# EPICS autosave request: FOFBApp/Db/FOFBRtm_settings.req
$(P)$(R)RtmLampDacDataFromWb-SP
$(P)$(R)RtmLampAmpEn$(RTM_CHAN)-SP
$(P)$(R)RtmLampPIOLTriangEn$(RTM_CHAN)-SP
$(P)$(R)RtmLampPIOLSquareEn$(RTM_CHAN)-SP
$(P)$(R)RtmLampPISPSquareEn$(RTM_CHAN)-SP
$(P)$(R)RtmLampPIEn$(RTM_CHAN)-SP
$(P)$(R)RtmLampDacData$(RTM_CHAN)-SP
$(P)$(R)RtmLampDacWr$(RTM_CHAN)-SP
$(P)$(R)RtmLampPIKP$(RTM_CHAN)-SP
$(P)$(R)RtmLampPITI$(RTM_CHAN)-SP
$(P)$(R)RtmLampPISP$(RTM_CHAN)-SP
$(P)$(R)RtmLampPIOLDacCntMax-SP
$(P)$(R)RtmLampPISPLimInf-SP
$(P)$(R)RtmLampCurrentGain$(RTM_CHAN)-SP
$(P)$(R)RtmLampCurrentOffset$(RTM_CHAN)-SP
